FUNCTION_BLOCK FB_File
VAR_INPUT
END_VAR
VAR_OUTPUT
END_VAR
VAR
	fbFileOpen : FB_FileOpen;
	fbFileClose : FB_FileClose;
	fbFileLoad : FB_FileLoad;
	fileBuffer : ARRAY[0..99] OF BYTE;
END_VAR

fbFileLoad(
	sNetId:= , 
	sPathName:= 'c:\TEMP\LOG.txt', 
	pReadBuff:= ADR(fileBuffer), 
	cbReadLen:= SIZEOF(fileBuffer), 
	bExecute:= , 
	tTimeout:= , 
	bBusy=> , 
	bError=> , 
	nErrId=> , 
	cbRead=> );

END_FUNCTION_BLOCK

(* stored: Version 1.1.0.1, ProductVersion 3.1.4024.12
   POU FB_File: Id {4b87f0fb-3446-4e32-bd0a-78e268c1e56e}, SpecialFunc None *)
